FUNCTION_BLOCK SS5b_Camera (* Basic FB with empty ECC *)
  (* Standard: 61499-2 *)
  (* Version 1.0, 2024-10-03, DEVIASH *)
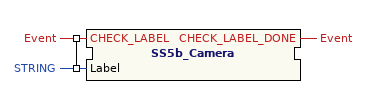
  EVENT_INPUT
    CHECK_LABEL WITH Label;
  END_EVENT
  EVENT_OUTPUT
    CHECK_LABEL_DONE;
  END_EVENT
  VAR_INPUT
    Label : STRING;
  END_VAR
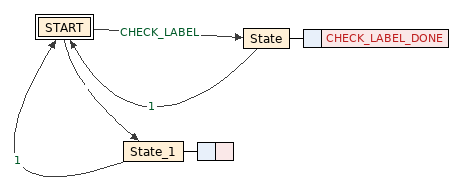
  EC_STATES
    START; (* Initial State *)
    State : -> CHECK_LABEL_DONE;
    State_1;
  END_STATES
  EC_TRANSITIONS
    START TO State := CHECK_LABEL;
    State TO START := 1;
    START TO State_1 := ;
    State_1 TO START := 1;
  END_TRANSITIONS
END_FUNCTION_BLOCK
